{attribute 'global_init_slot' := '1'}
VAR_GLOBAL
	
	StartCycle AT %I*: BOOL;
	StartCycle_HMI : BOOL;
	StopCycle AT %I*: BOOL;
	StopCycle_HMI : BOOL;
	ResetSafety AT %I*: BOOL;

    RTrigStart : R_TRIG;
    RTrigStop  : R_TRIG;

    bStartCycleMem : BOOL;  
    bStopCycleMem  : BOOL;  
	
	SafetyRelayStatus AT %I*: BOOL;
	
	gSystemAlarmStatus : ST_SystemAlarmStatus;
	
	PLC_Fan_Steppers AT %I*: BOOL;
	
	CONTROL : BOOL := FALSE;
	
	Result          : INT := 0;
	
	sRequestedActuator : STRING := '';
	bIsPoweredUp     : ARRAY[1..4] OF BOOL;
	
	aLookupTable : ARRAY[1..100] OF ST_LookupEntry := [
		(nX := 1, sY := 'Chariot', sValue := ADR(Tri1_Mot_FB), sCommand := ADR(Tri1_Mot_Cmd)),
		(nX := 1, sY := 'Compressor', sValue := ADR(Cmp1_Mot_FB), sCommand := ADR(Cmp1_Mot_Cmd)),
		(nX := 1, sY := 'Sensor', sValue := ADR(Piv1_Mot_FB), sCommand := ADR(Piv1_Mot_Cmd)),
		(nX := 2, sY := 'Chariot', sValue := ADR(Tri2_Mot_FB), sCommand := ADR(Tri2_Mot_Cmd)),
		(nX := 3, sY := 'HeatExCoupola', sValue := ADR(Gui1_Mot_FB), sCommand := ADR(Gui1_Mot_Cmd)),
		(nX := 3, sY := 'RegenCoupola', sValue := ADR(Gui2_Mot_FB), sCommand := ADR(Gui2_Mot_Cmd)),
		(nX := 3, sY := 'Chariot', sValue := ADR(Tri3_Mot_FB), sCommand := ADR(Tri3_Mot_Cmd)),
		(nX := 3, sY := 'Compressor', sValue := ADR(Cmp2_Mot_FB), sCommand := ADR(Cmp2_Mot_Cmd)),
		(nX := 4, sY := 'Chariot', sValue := ADR(Tri4_Mot_FB), sCommand := ADR(Tri4_Mot_Cmd)),
		(nX := 1, sY := 'Home', sValue := ADR(Rail1_Mot_FB), sCommand := ADR(Rail1_Mot_Cmd)),
		(nX := 1, sY := 'SetHome', sValue := ADR(Rail1_Mot_FB), sCommand := ADR(Rail1_Mot_Cmd)),
		(nX := 1, sY := 'Motor', sValue := ADR(Rail1_Mot_FB), sCommand := ADR(Rail1_Mot_Cmd)),
		(nX := 2, sY := 'Home', sValue := ADR(Rail2_Mot_FB), sCommand := ADR(Rail2_Mot_Cmd)),
		(nX := 2, sY := 'SetHome', sValue := ADR(Rail2_Mot_FB), sCommand := ADR(Rail2_Mot_Cmd)),
		(nX := 2, sY := 'Motor', sValue := ADR(Rail2_Mot_FB), sCommand := ADR(Rail2_Mot_Cmd)),
		(nX := 3, sY := 'Home', sValue := ADR(Rail3_Mot_FB), sCommand := ADR(Rail3_Mot_Cmd)),
		(nX := 3, sY := 'SetHome', sValue := ADR(Rail3_Mot_FB), sCommand := ADR(Rail3_Mot_Cmd)),
		(nX := 3, sY := 'Motor', sValue := ADR(Rail3_Mot_FB), sCommand := ADR(Rail3_Mot_Cmd)),
		(nX := 4, sY := 'Home', sValue := ADR(Rail4_Mot_FB), sCommand := ADR(Rail4_Mot_Cmd)),
		(nX := 4, sY := 'SetHome', sValue := ADR(Rail4_Mot_FB), sCommand := ADR(Rail4_Mot_Cmd)),
		(nX := 4, sY := 'Motor', sValue := ADR(Rail4_Mot_FB), sCommand := ADR(Rail4_Mot_Cmd))
	];
    nEntryCount : INT := 21; 
END_VAR

(* stored: Version 1.1.0.1, ProductVersion 3.1.4026.11
   GVL GVL: Id {84031c49-9b58-4990-8455-46264bcb9bf2} *)
